// TIA Portal V21 export
TYPE "udt_TEST"
   STRUCT
      "a" : Bool;
   END_STRUCT;
END_TYPE
